# EPICS substitutions: elioApp/Db/EL3314.substitutions
file EL3314.template { pattern
{ CHAN	}
{ 1	}
{ 2	}
{ 3	}
{ 4	}
}
